TYPE E_Terminals :
(
	TempSens1,
	TempSens2,
	TempSens3,
	TempSens3Wire,
	PressSens,
	PowMeasTerm,
	AnalogOutp,
	OutpSwitchValv,
	OutpCont
);
END_TYPE

(* stored: Version 1.1.0.1, ProductVersion 3.1.4018.2
   DUT E_Terminals: Id {0883c50c-4f56-420c-b099-505669e99866} *)
